FUNCTION_BLOCK FB_RampVelo
VAR_INPUT
	bExecute:BOOL;
	fVelSetIn:LREAL:=0;
	iBlockSampleTimeMicroS:INT:=10000;
	fVelActIn:LREAL:=0;
END_VAR
VAR_IN_OUT
    fVelSetOut:LREAL:=0;
END_VAR
VAR
  fChangePerCycle:LREAL:=0;
  fCurrAcc:LREAL:=0;
  fAccX1:LREAL:=0.8;
  fAccX2:LREAL:=0.99;
  fAccY1:LREAL:=GVL_Parameters.fAccDefaultVel;
  fAccY2:LREAL:=GVL_Parameters.fAccDefaultVel*0.1;
  fAccK:LREAL:=0;
  fAccM:LREAL:=0;
  x:LREAL:=0;
  bExecuteOld:BOOL:=FALSE;
  fActVeloOld:LREAL:=0;  // Used for extra sanity check of velo
END_VAR

// Function: Ramp velocity with a defined acceleration.
// Accelerartion is ramped down when apparching velosity setpoint in order to reduce
// overshoot and oscillations..
// Author: Anders Sandström 20200114

IF NOT bExecute OR ABS(fVelSetIn) > GVL_Parameters.fMaximumSPeedSPRpm THEN
  fVelSetOut:=0;
  bExecuteOld:=bExecute;
  fActVeloOld:=fVelActIn;
  RETURN;
END_IF;

// Start at current velocity if retreigger (avoid go to zero)
IF NOT bExecuteOld AND bExecute THEN
  // Sanity check of the actual velocity
  IF fVelActIn > -GVL_Parameters.fMaximumSPeedRpm AND 
	 fVelActIn < GVL_Parameters.fMaximumSPeedRpm AND 
	 fActVeloOld > -GVL_Parameters.fMaximumSPeedRpm AND 
	 fActVeloOld < GVL_Parameters.fMaximumSPeedRpm THEN
	fVelSetOut:=(fVelActIn+fActVeloOld)/2;  //Set to average of two cycles
  ELSE
    fVelSetOut:=0;
  END_IF  
END_IF
bExecuteOld:=bExecute;
fActVeloOld:=fVelActIn;

IF fVelSetOut=fVelSetIn THEN
  fVelSetOut:=fVelSetIn;
  RETURN;
END_IF;

//Reduce overshoot by lowering acc when closing in on setpoint (linear)
//           Acceleration [rpm/s^2]
//                 ^
//  y1=defAcc     -|-----------------\
//                 |                  \  
//                 |                   \
//                 |                    \ 
//                 |                     \
//  y2=defAcc*0.1 -|                      \-----------------
//                 |--------------------------------------------> fSetOut/fSetIn []
//                                 x1=0.8 x2=1.0 

fAccK:=(fAccY2-fAccY1)/(fAccX2-fAccX1);
fAccM:= fAccY1-fAccK*fAccX1;
IF fVelSetIn<>0 THEN
  x:=fVelSetOut/fVelSetIn;
ELSE
  x:=1.0;
END_IF
// try linear ramp down off acceleration from 0.8*velsetin to velset in (from defacc to 0.1* defacc)
fCurrAcc:=GVL_Parameters.fAccDefaultVel;
IF fVelSetIn > fVelSetOut THEN 
  IF x > fAccX1 AND x <= fAccX2 AND fVelSetOut<fVelSetIn THEN
    fCurrAcc:=fAccK*fVelSetOut/fVelSetIn+fAccM;
  ELSIF x >= fAccX2 THEN
    fCurrAcc:=GVL_Parameters.fAccDefaultVel*0.1;
  END_IF
END_IF

// Change per execution
fChangePerCycle:=fCurrAcc/(1E6/iBlockSampleTimeMicroS);

// Ramp finished
IF ABS(fVelSetIn-fVelSetOut)<fChangePerCycle THEN
  fVelSetOut:=fVelSetIn;
  RETURN;
END_IF

//Acc
IF fVelSetIn > fVelSetOut THEN             // Acc
  fVelSetOut:=fVelSetOut+fChangePerCycle;
ELSIF fVelSetIn < fVelSetOut THEN          // Dec
  fVelSetOut:=fVelSetOut-fChangePerCycle;
END_IF

END_FUNCTION_BLOCK

(* stored: Version 1.1.0.1, ProductVersion 3.1.4024.6
   POU FB_RampVelo: Id {d4ab285d-06ec-4c4c-adcf-b2df350d8b46}, SpecialFunc None *)
